DEVICE_TYPE TESTPAR_DEV (* Test Java initialization of parameters in Device Type *)
  (* Standard: 61499-1 *)
  (* Version 0.0, 2004-12-16, JHC, Rockwell Automation *)
  (* Compiler header: package fb.rt.test; *)
  (* Compiler Java Sun JDK 1.4.2 *)
  VAR_INPUT
    PUBL_ID : WSTRING;
  END_VAR
  RESOURCE RES1 : TESTPAR_RES(SUBSC_ID := "225.0.0.1:1025")
  END_RESOURCE
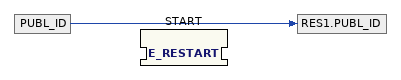
  FBS
    START : E_RESTART;
  END_FBS
  DATA_CONNECTIONS
    PUBL_ID TO RES1.PUBL_ID;
  END_CONNECTIONS
END_DEVICE_TYPE
